// TwinCAT 3 PLC project Main
// ProgramVersion: 3.1.4023.0
// libraries:
//   Tc2_Standard, * (Beckhoff Automation GmbH)
//   Tc2_System, * (Beckhoff Automation GmbH)
//   Tc3_JsonXml, * (Beckhoff Automation GmbH)
//   Tc3_Module, * (Beckhoff Automation GmbH)
//   Tc3_Vision, * (Beckhoff Automation GmbH)
// project tree:
//   / PlcTask.TcTTO
//   POUs/ MAIN.TcPOU
// real-time tasks:
//   TASK PlcTask: cycle T#10ms, priority 20, ADS port 350

CONFIGURATION Main
    RESOURCE PLC ON TwinCAT3
        TASK PlcTask(INTERVAL := T#10ms, PRIORITY := 20);
        PROGRAM MAIN WITH PlcTask : MAIN;
    END_RESOURCE
END_CONFIGURATION

// ---- POUs/MAIN.TcPOU
PROGRAM MAIN
VAR
	readImage: FB_VN_ReadImage;
	myImage : ITcVnImage;
	hr : HRESULT;	
	exportImageSize: ULINT;
	result : STRING;
	buffer : POINTER TO BYTE;
	jsonDocument : FB_JsonSaxWriter;
	jsonString : STRING(5000000);
	myDisplayableImage : ITcVnDisplayableImage;
END_VAR
VAR CONSTANT
	MAX_UDINT : UDINT := 4294967295;
END_VAR

readImage(
    sFilePath := 'C:\temp\image.png', 
    ipDestImage := myImage,
    bRead := TRUE,
    nTimeout := T#20S
);

IF readImage.bBusy OR readImage.bError OR myImage = 0 THEN
    RETURN;
END_IF

result := 'Start';

hr := F_VN_ExportImageAsBmpSize(ipImage:=myImage,nBufferSize:=exportImageSize,hrPrev:=hr);

IF Failed(hr) THEN
	result := 'Unable to convert as size check failed';
	RETURN;
END_IF

IF exportImageSize > MAX_UDINT THEN
	result := 'Unable to convert as image is too big.  Use a premade byte array instead';
	RETURN;
END_IF

IF exportImageSize <= 0 THEN
	result := 'Unable to convert as image is empty';
	RETURN;
END_IF
	
buffer := __NEW(BYTE,ULINT_TO_UDINT(exportImageSize));
hr := F_VN_ExportImageAsBmp(ipImage:=myImage,pBuffer:=buffer,nBufferSize:=exportImageSize,hrPrev:=hr);

IF FAILED(hr) THEN
	result := 'Export failed';
	__DELETE(buffer);
	RETURN;
END_IF

jsonDocument.ResetDocument();
jsonDocument.StartObject();
jsonDocument.AddKeyString('mime','image/bmp');
jsonDocument.AddKey('data');
jsonDocument.AddBase64(buffer,ULINT_TO_DINT(exportImageSize));
jsonDocument.EndObject();
jsonDocument.CopyDocument(jsonString,SIZEOF(jsonString));

result := 'Success';

__DELETE(buffer);

hr := F_VN_TransformIntoDisplayableImage(myImage, myDisplayableImage, S_OK);

END_PROGRAM
